FUNCTION_BLOCK BUBBLESIZEGEN (* level based bubble size generator *)
  (* Version 1.0, AN, SWDC RTSoft *)
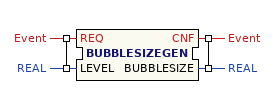
  EVENT_INPUT
    REQ WITH LEVEL;
  END_EVENT
  EVENT_OUTPUT
    CNF WITH BUBBLESIZE;
  END_EVENT
  VAR_INPUT
    LEVEL : REAL;
  END_VAR
  VAR_OUTPUT
    BUBBLESIZE : REAL;
  END_VAR
END_FUNCTION_BLOCK
